{attribute addProperty BoxType "EL3602-0002-0016"}
{attribute addProperty Id "AI_Inputs_ChannelAT %I*ARRAY[0..1] OF AI_Inputs_Channel_BED3E98C96120WcStateAT %I*WcState_F855686C1620InfoDataAT %I*InfoData_BC63D37F80100"}
{attribute addProperty CRC "2822285772"}
{attribute addProperty SizeInBites "192"}
{attribute addProperty SizeInBytes "24"}
TYPE EL3602_48691765 :
STRUCT
	{attribute addProperty Name "AI_Inputs_Channel"}
	AI_Inputs_Channel : ARRAY[0..1] OF AI_Inputs_Channel_BED3E98C;
	{attribute addProperty Name "WcState"}
	WcState : WcState_F855686C;
	{attribute addProperty Name "InfoData"}
	InfoData : InfoData_BC63D37F;
END_STRUCT
END_TYPE

(* stored: Version 1.2.0.0, ProductVersion 3.1.4024.9
   DUT EL3602_48691765: Id {4db6af9f-b1b7-4d8b-9359-37ee56219c02} *)
